// TIA Portal V18 export
FUNCTION "AHU_EqpCtrl" : Void   // FC60300, FBD
{ S7_Optimized_Access := 'TRUE' }
VERSION : 0.1
// stored: AutoNumber false, IsIECCheckEnabled false, SetENOAutomatically false, UDAEnableTagReadback false
   VAR_INPUT
      iUnitID : Int;   // 1=AHUFood, 2=AHUNonFood
   END_VAR
   VAR_TEMP
      FA_temp : Real;
   END_VAR
BEGIN

REGION Network 1: Forming Eqp State with respect of Season and Actual State
   // 0 = Winter
   // 1= Summer
   // 2=Midseason
   // 3=Auto
   // 
   // "HVAC".Season.Actual
   // 0 = Winter
   // 1=Summer
   // 2=Midseason
   // 3=Auto
   // 
   // Type                                             Control State
   // 0 = no ctrl                                             0 = Stopped/Closed/NA
   // 1 = Proxi/Adaptation                           1 = 100%/FullyOpened/ 
   // 2=                                                           2 = RegulationEnable
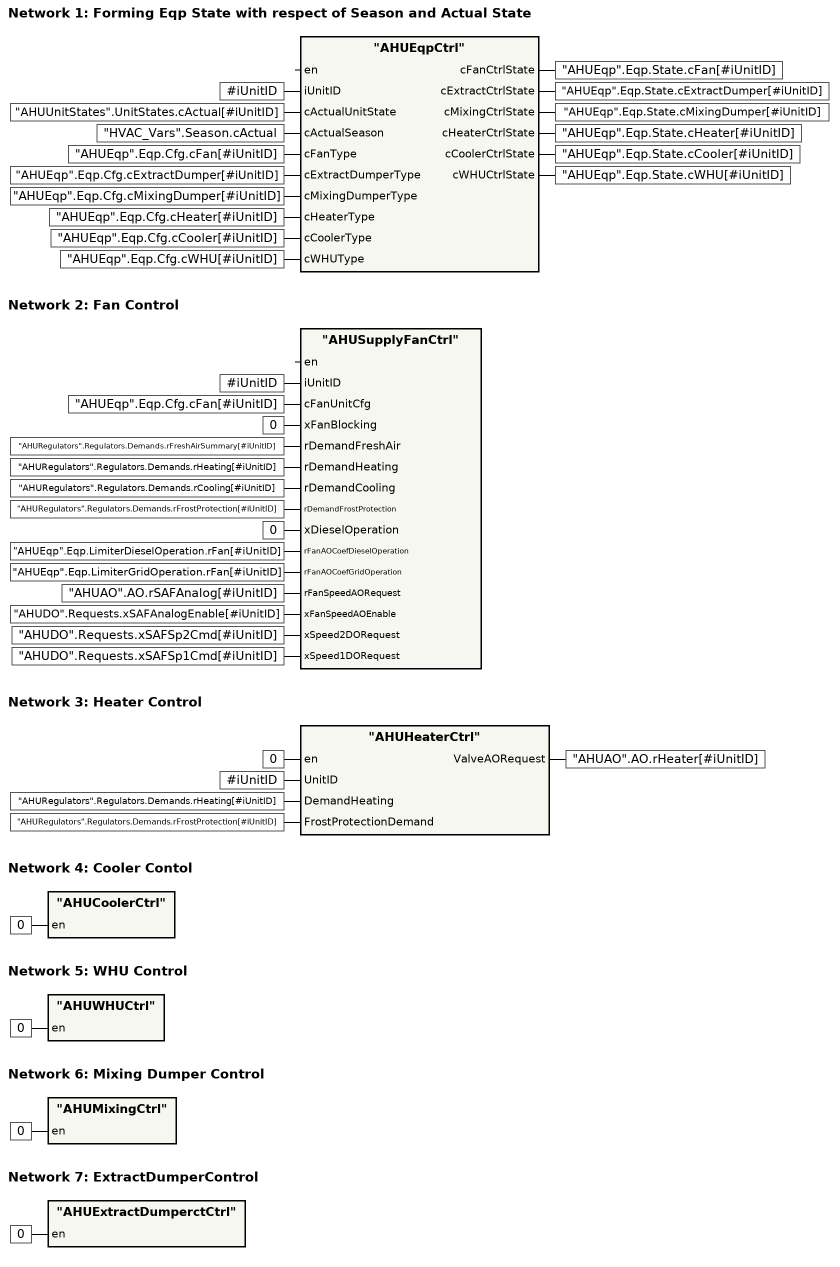
   "AHUEqpCtrl"(iUnitID := #iUnitID,
                cActualUnitState := "AHUUnitStates".UnitStates.cActual[#iUnitID],
                cActualSeason := "HVAC_Vars".Season.cActual,
                cFanType := "AHUEqp".Eqp.Cfg.cFan[#iUnitID],
                cExtractDumperType := "AHUEqp".Eqp.Cfg.cExtractDumper[#iUnitID],
                cMixingDumperType := "AHUEqp".Eqp.Cfg.cMixingDumper[#iUnitID],
                cHeaterType := "AHUEqp".Eqp.Cfg.cHeater[#iUnitID],
                cCoolerType := "AHUEqp".Eqp.Cfg.cCooler[#iUnitID],
                cWHUType := "AHUEqp".Eqp.Cfg.cWHU[#iUnitID],
                cFanCtrlState => "AHUEqp".Eqp.State.cFan[#iUnitID],
                cExtractCtrlState => "AHUEqp".Eqp.State.cExtractDumper[#iUnitID],
                cMixingCtrlState => "AHUEqp".Eqp.State.cMixingDumper[#iUnitID],
                cHeaterCtrlState => "AHUEqp".Eqp.State.cHeater[#iUnitID],
                cCoolerCtrlState => "AHUEqp".Eqp.State.cCooler[#iUnitID],
                cWHUCtrlState => "AHUEqp".Eqp.State.cWHU[#iUnitID]);
END_REGION

REGION Network 2: Fan Control
   "AHUSupplyFanCtrl"(iUnitID := #iUnitID,
                      cFanUnitCfg := "AHUEqp".Eqp.Cfg.cFan[#iUnitID],
                      xFanBlocking := 0,
                      rDemandFreshAir := "AHURegulators".Regulators.Demands.rFreshAirSummary[#iUnitID],
                      rDemandHeating := "AHURegulators".Regulators.Demands.rHeating[#iUnitID],
                      rDemandCooling := "AHURegulators".Regulators.Demands.rCooling[#iUnitID],
                      rDemandFrostProtection := "AHURegulators".Regulators.Demands.rFrostProtection[#iUnitID],
                      xDieselOperation := 0,
                      rFanAOCoefDieselOperation := "AHUEqp".Eqp.LimiterDieselOperation.rFan[#iUnitID],
                      rFanAOCoefGridOperation := "AHUEqp".Eqp.LimiterGridOperation.rFan[#iUnitID],
                      rFanSpeedAORequest := "AHUAO".AO.rSAFAnalog[#iUnitID],
                      xFanSpeedAOEnable := "AHUDO".Requests.xSAFAnalogEnable[#iUnitID],
                      xSpeed2DORequest := "AHUDO".Requests.xSAFSp2Cmd[#iUnitID],
                      xSpeed1DORequest := "AHUDO".Requests.xSAFSp1Cmd[#iUnitID]);
END_REGION

REGION Network 3: Heater Control
   IF 0 THEN
       "AHUHeaterCtrl"(UnitID := #iUnitID,
                       DemandHeating := "AHURegulators".Regulators.Demands.rHeating[#iUnitID],
                       FrostProtectionDemand := "AHURegulators".Regulators.Demands.rFrostProtection[#iUnitID],
                       ValveAORequest => "AHUAO".AO.rHeater[#iUnitID]);
   END_IF;
END_REGION

REGION Network 4: Cooler Contol
   IF 0 THEN "AHUCoolerCtrl"(); END_IF;
END_REGION

REGION Network 5: WHU Control
   IF 0 THEN "AHUWHUCtrl"(); END_IF;
END_REGION

REGION Network 6: Mixing Dumper Control
   IF 0 THEN "AHUMixingCtrl"(); END_IF;
END_REGION

REGION Network 7: ExtractDumperControl
   IF 0 THEN "AHUExtractDumperctCtrl"(); END_IF;
END_REGION
END_FUNCTION
